Universal Robots PolyScope program: string_waypoints.urp

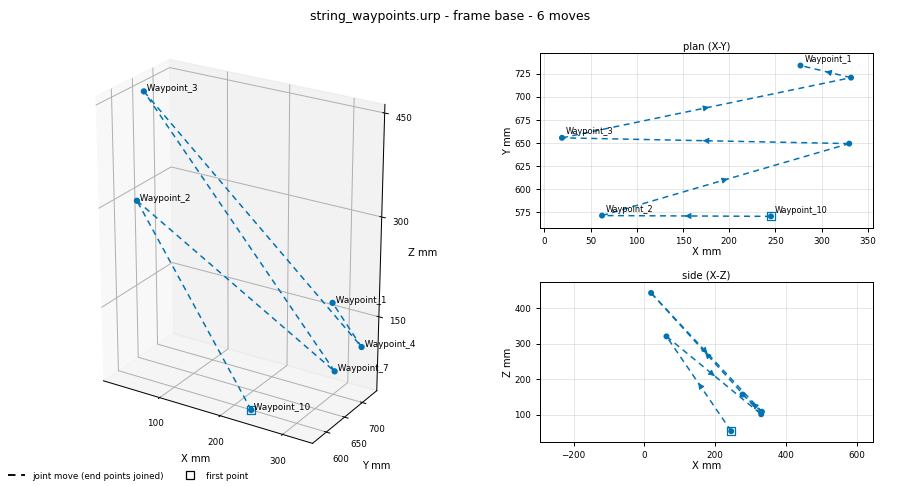
[picture p0: tool path of string_waypoints.urp in frame base, 6 of 6 moves have a stored position in this frame; points joined in program order, loops and branches not executed]
Program string_waypoints (installation=string_planes directory=/programs createdIn=5.17.3 lastSavedIn=5.17.3 robotSerialNumber=20245501435)
Calibrated DH parameters: a=[0.000154, -0.137004, -0.385524, -0.00002, 0.000092, 0]; d=[0.162441, 211.794786, -230.585024, 18.923638, 0.099786, 0.09951]; alpha=[1.569493, -0.001902, 0.003874, 1.570111, -1.570167, 0]; deltaTheta=[0, -1.242934, 1.056292, 0.186646, 0.000002, 0.000001]
InitVariablesNode
Robot Program (runOnlyOnce=false)
  MoveJ speed 60 deg/s, acceleration 80 deg/s^2 (useActiveTCP=true) feature=Base
    Waypoint Waypoint_10: TCP in base x=245.284 y=570.71 z=53.266 mm, rx=-1.8425 ry=-1.3918 rz=0.0687 rad; joints [-132.226, -24.798, 96.314, -169.322, -42.692, -112.607] deg; TCP offset x=28.21 y=-96.107 z=-99.69 mm, rx=0 ry=0 rz=0 rad
    Waypoint Waypoint_2: TCP in base x=62.353 y=571.559 z=321.201 mm, rx=-1.5659 ry=-1.6472 rz=0.323 rad; joints [-116.09, -61.712, 109.823, -138.497, -38.878, -118.568] deg; TCP offset x=28.21 y=-96.107 z=-99.69 mm, rx=0 ry=0 rz=0 rad
  MoveJ speed 60 deg/s, acceleration 80 deg/s^2 (useActiveTCP=true) feature=Base
    Waypoint Waypoint_7: TCP in base x=329.981 y=649.486 z=101.065 mm, rx=-1.7033 ry=-1.7268 rz=0.636 rad; joints [-132.743, -28.556, 74.955, -104.888, -53.814, -143.829] deg
    Waypoint Waypoint_3: TCP in base x=18.957 y=655.733 z=443.885 mm, rx=-1.6477 ry=-1.7733 rz=0.627 rad; joints [-109.658, -66.048, 89.298, -99.16, -44.965, -119.608] deg
  MoveJ speed 60 deg/s, acceleration 80 deg/s^2 (useActiveTCP=true) feature=Base
    Waypoint Waypoint_4: TCP in base x=331.973 y=720.894 z=108.291 mm, rx=-1.645 ry=-2.1081 rz=1.0591 rad; joints [-129.773, -21.651, 52.373, -76.468, -76.907, -149.022] deg
  MoveJ speed 60 deg/s, acceleration 80 deg/s^2 (useActiveTCP=true) feature=Base
    Waypoint Waypoint_1: TCP in base x=277.237 y=734.032 z=156.892 mm, rx=1.7389 ry=2.3104 rz=-1.1078 rad; joints [-126.647, -28.123, 54.729, -74.616, -91.964, -141.812] deg; TCP offset x=28.21 y=-96.107 z=-99.69 mm, rx=0 ry=0 rz=0 rad
